TYPE ST_Recipe :
	STRUCT
		ValueA : LREAL;
		ValueB : DINT;
		ValueC : BOOL;
	END_STRUCT
END_TYPE

(* stored: Version 1.1.0.1, ProductVersion 3.1.4026.18
   DUT ST_Recipe: Id {c77a914c-cc7f-43a9-980c-817d2abb092c} *)
